Fanuc KAREL source: NC0065.KL

-- PROVISIONAL review KL for V770-1; original PC SHA256 3a997e2fa4e70be138acc6d0913616bf1ffe66972a29a7fd5242a80901d41405
-- Incomplete behavior may be omitted. Consult companion uncertainty JSON. Do not deploy.
PROGRAM NC0065
%NOLOCKGROUP
-- UNRESOLVED_LOCAL_POOL 6 cells at code offset 3; source declarations unknown
-- DIRECT_LOCAL_WORD_ACCESS alone does not prove INTEGER, REAL, or BOOLEAN
BEGIN
  -- UNRESOLVED_PC offsets 0-8; opcodes 2B,2C,7B
  -- UNRESOLVED_PC offsets 13-20; opcodes 9D,23
  -- UNRESOLVED_PC offsets 25-54; opcodes 9D,23,9E,2E,22,7A
  -- UNRESOLVED_PC offsets 59-88; opcodes 9D,23,9E,2E,22,7A
  -- UNRESOLVED_PC offsets 93-122; opcodes 9D,23,9E,2E,22,7A
  -- UNRESOLVED_PC offsets 127-156; opcodes 9D,23,9E,2E,22,7A
  -- UNRESOLVED_PC offsets 161-190; opcodes 9D,23,9E,2E,22,7A
  -- UNRESOLVED_PC offsets 195-209; opcodes 21,9D,52,23
  -- UNRESOLVED_PC offsets 214-229; opcodes 20,2C,23
  -- UNRESOLVED_PC offsets 234-249; opcodes 20,2C,23
  -- UNRESOLVED_PC offsets 254-269; opcodes 20,2C,23
  -- UNRESOLVED_PC offsets 274-289; opcodes 20,2C,23
  -- UNRESOLVED_PC offsets 294-309; opcodes 20,2C,23
  -- UNRESOLVED_PC offsets 314-318; opcodes 7F
  -- UNRESOLVED_PC offsets 323-327; opcodes 27,AA
  -- UNRESOLVED_PC offsets 332-336; opcodes 7F
END NC0065
